(* IEC 61131-3 sources: json/src/Properties, 3 files *)

(* ---- DoubleInt.st ---- *)
USING Simatic.Ax.Conversion;

NAMESPACE Simatic.Ax.Json.Properties
    CLASS DoubleInt EXTENDS JsonNumber
        VAR PUBLIC
            value : DINT;
        END_VAR

        METHOD PUBLIC OVERRIDE ToString : STRING
            ToString := THIS.ToStringHelper(Integer.ToString(value := value));
        END_METHOD
    END_CLASS
END_NAMESPACE

(* ---- JsonNumber.st ---- *)
USING System.Strings;

NAMESPACE Simatic.Ax.Json
    CLASS JsonNumber EXTENDS JsonProperty

        METHOD PROTECTED OVERRIDE ToStringHelper : STRING
            VAR_INPUT
                valueAsString : STRING;
            END_VAR
            VAR_TEMP
                _str : STRING;
            END_VAR
            _str := Concat('"', key, '": ', valueAsString);
            ToStringHelper := _str;
        END_METHOD

        METHOD PUBLIC OVERRIDE ToString : STRING
            ;
        END_METHOD
    END_CLASS
END_NAMESPACE

(* ---- JsonProperty.st ---- *)
USING System.Strings;

NAMESPACE Simatic.Ax.Json
    CLASS ABSTRACT JsonProperty IMPLEMENTS IJsonObject
        VAR PUBLIC
            key : STRING;
        END_VAR

        VAR PROTECTED
            _next : IJsonObject;
        END_VAR

        METHOD PUBLIC ABSTRACT ToString : STRING
        END_METHOD

        METHOD PUBLIC Serialize : BOOL
            VAR_INPUT
                t : ARRAY [*] OF BYTE;
            END_VAR
            ;
        END_METHOD

        METHOD PROTECTED ToStringHelper : STRING
            VAR_INPUT
                valueAsString : STRING;
            END_VAR
            VAR_TEMP
                _str : STRING;
            END_VAR
            _str := Concat('"', key, '"', ': "');
            _str := Concat(_str, valueAsString, '"');
            ToStringHelper := _str;
        END_METHOD

        METHOD PUBLIC HasNext : BOOL
            HasNext := _next <> NULL;
        END_METHOD

        METHOD PUBLIC GetNext : IJsonObject
            GetNext := _next;
        END_METHOD

        METHOD PUBLIC AddObject
            VAR_INPUT
                obj : IJsonObject;
            END_VAR
            _next := obj;
        END_METHOD

    END_CLASS
END_NAMESPACE
